// TIA Portal project "Forno" (V14)

(* hardware
DEVICE "S7-1200 station_1"  S7-1200 Station
   slot 0: "Rack_0"  Rack  V1.0
   slot 1: "PLC_1"  CPU 1214C DC/DC/DC  6ES7 214-1AG31-0XB0  V3.0
*)

// ===== PLC "PLC_1"  CPU 1214C DC/DC/DC =====

VAR_GLOBAL   // PLC tag table "Default tag table"
   "Pressostato_alta" AT %M0.0 : Bool;
   "Pressostato_baixa" AT %M0.1 : Bool;
   "Fluxo_exaust" AT %M0.2 : Bool;
   "Fluxo_forc" AT %M0.3 : Bool;
   "porta_closed" AT %M0.4 : Bool;
   "porta_opened" AT %M0.5 : Bool;
   "chama_piloto" AT %M0.6 : Bool;
   "chama_pricipal" AT %M0.7 : Bool;
   "Relay_chama_ok" AT %M1.0 : Bool;
   "Vent_exaust" AT %Q0.0 : Bool;
   "Vent_forc" AT %Q0.1 : Bool;
   "open_porta" AT %Q0.2 : Bool;
   "close_porta" AT %Q0.3 : Bool;
   "Valv_controle" AT %Q0.4 : Bool;
   "Bloqueio" AT %Q0.5 : Bool;
   "Relay_chama_comando" AT %Q0.6 : Bool;
   "intertravamentos" AT %M1.1 : Bool;
   "botao_on" AT %M1.2 : Bool;
   "partida_ok" AT %M1.3 : Bool;
   "purga_ok" AT %M1.4 : Bool;
   "ignicao" AT %M1.6 : Bool;
   "tentativa1" AT %M1.7 : Bool;
   "tentativa2" AT %M2.0 : Bool;
   "tentativa3" AT %M2.1 : Bool;
END_VAR

// folder: System blocks/Program resources

DATA_BLOCK "IEC_Timer_0_DB"   // DB1
{ S7_Optimized_Access := 'TRUE' }
AUTHOR : Simatic
FAMILY : IEC
NAME : IEC_TMR
VERSION : 1.0
// stored: InstanceOfName IEC_TIMER
"IEC_TIMER"
BEGIN
END_DATA_BLOCK

DATA_BLOCK "IEC_Timer_0_DB_1"   // DB2
{ S7_Optimized_Access := 'TRUE' }
AUTHOR : Simatic
FAMILY : IEC
NAME : IEC_TMR
VERSION : 1.0
// stored: InstanceOfName IEC_TIMER
"IEC_TIMER"
BEGIN
END_DATA_BLOCK

DATA_BLOCK "IEC_Timer_0_DB_3"   // DB4
{ S7_Optimized_Access := 'TRUE' }
AUTHOR : Simatic
FAMILY : IEC
NAME : IEC_TMR
VERSION : 1.0
// stored: InstanceOfName IEC_TIMER
"IEC_TIMER"
BEGIN
END_DATA_BLOCK

DATA_BLOCK "IEC_Timer_0_DB_4"   // DB5
{ S7_Optimized_Access := 'TRUE' }
AUTHOR : Simatic
FAMILY : IEC
NAME : IEC_TMR
VERSION : 1.0
// stored: InstanceOfName IEC_TIMER
"IEC_TIMER"
BEGIN
END_DATA_BLOCK

// folder: (top level)

FUNCTION "Purga" : Void   // FC1, LAD
{ S7_Optimized_Access := 'TRUE' }
VERSION : 0.1
BEGIN

REGION Network 1
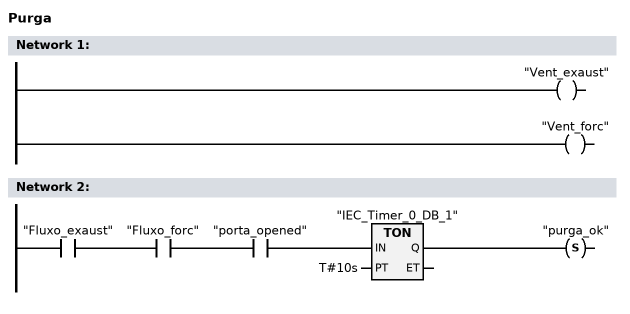
   RUNG wire#powerrail
      Coil( "Vent_exaust" )
   END_RUNG
   RUNG wire#powerrail
      Coil( "Vent_forc" )
   END_RUNG
   // the same network as SCL:
   "Vent_exaust" := TRUE;
   "Vent_forc" := TRUE;
END_REGION

REGION Network 2
   "IEC_Timer_0_DB_1".TON(IN := "Fluxo_exaust" AND "Fluxo_forc" AND "porta_opened", PT := T#10s);
   IF "IEC_Timer_0_DB_1".Q THEN "purga_ok" := TRUE; END_IF;
END_REGION
END_FUNCTION

ORGANIZATION_BLOCK "Main"   // OB1, LAD, ProgramCycle
TITLE = "Main Program Sweep (Cycle)"
{ S7_Optimized_Access := 'TRUE' }
VERSION : 0.1
BEGIN

REGION Network 1
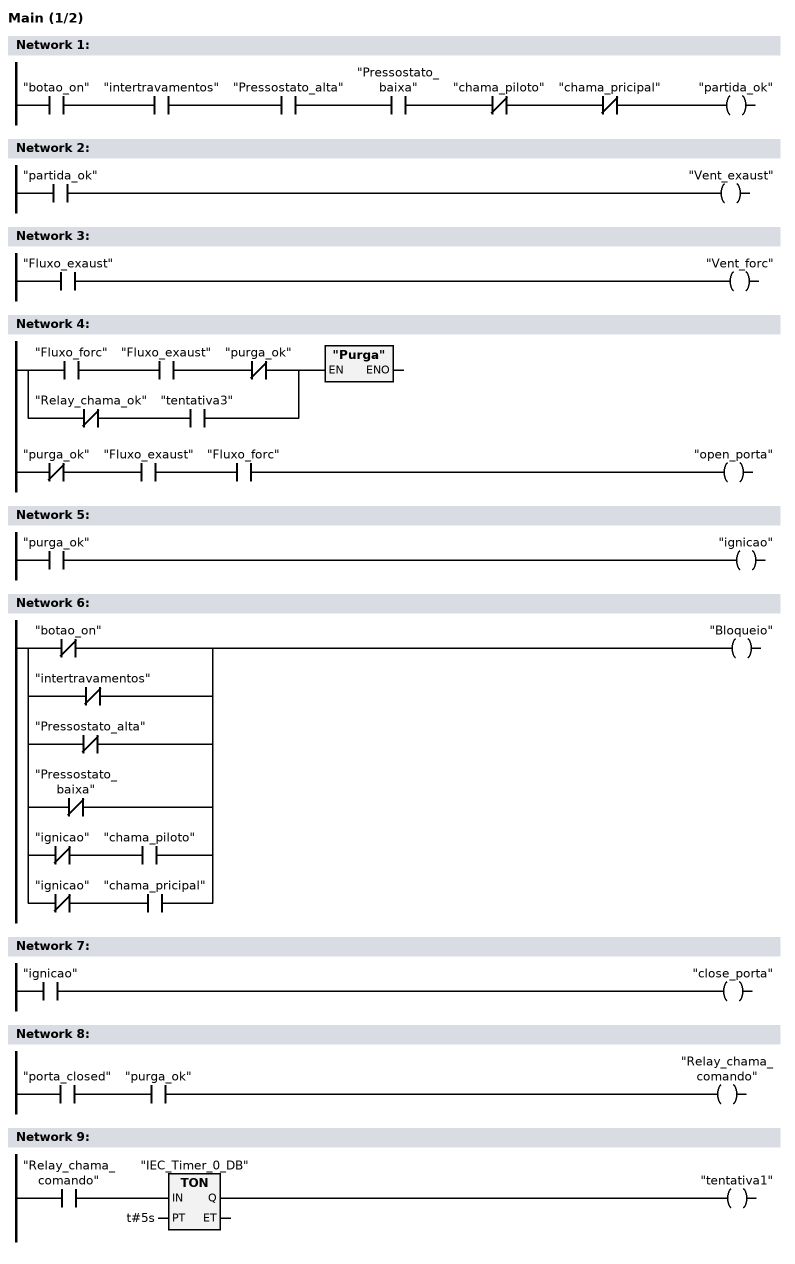
   RUNG wire#powerrail
      Contact( "botao_on" )
      Contact( "intertravamentos" )
      Contact( "Pressostato_alta" )
      Contact( "Pressostato_baixa" )
      I_Contact( "chama_piloto" )
      I_Contact( "chama_pricipal" )
      Coil( "partida_ok" )
   END_RUNG
   // the same network as SCL:
   "partida_ok" := "botao_on" AND "intertravamentos" AND "Pressostato_alta" AND "Pressostato_baixa" AND NOT "chama_piloto" AND NOT "chama_pricipal";
END_REGION

REGION Network 2
   RUNG wire#powerrail
      Contact( "partida_ok" )
      Coil( "Vent_exaust" )
   END_RUNG
   // the same network as SCL:
   "Vent_exaust" := "partida_ok";
END_REGION

REGION Network 3
   RUNG wire#powerrail
      Contact( "Fluxo_exaust" )
      Coil( "Vent_forc" )
   END_RUNG
   // the same network as SCL:
   "Vent_forc" := "Fluxo_exaust";
END_REGION

REGION Network 4
   RUNG wire#powerrail
      Contact( "Fluxo_forc" )
      Contact( "Fluxo_exaust" )
      I_Contact( "purga_ok" )
      wire#w1
      "Purga"()
   END_RUNG
   RUNG wire#powerrail
      I_Contact( "Relay_chama_ok" )
      Contact( "tentativa3" )
   END_RUNG wire#w1
   RUNG wire#powerrail
      I_Contact( "purga_ok" )
      Contact( "Fluxo_exaust" )
      Contact( "Fluxo_forc" )
      Coil( "open_porta" )
   END_RUNG
   // the same network as SCL:
   IF ("Fluxo_forc" AND "Fluxo_exaust" AND NOT "purga_ok") OR (NOT "Relay_chama_ok" AND "tentativa3") THEN
       "Purga"();
   END_IF;
   "open_porta" := NOT "purga_ok" AND "Fluxo_exaust" AND "Fluxo_forc";
END_REGION

REGION Network 5
   RUNG wire#powerrail
      Contact( "purga_ok" )
      Coil( "ignicao" )
   END_RUNG
   // the same network as SCL:
   "ignicao" := "purga_ok";
END_REGION

REGION Network 6
   RUNG wire#powerrail
      I_Contact( "botao_on" )
      wire#w1
      Coil( "Bloqueio" )
   END_RUNG
   RUNG wire#powerrail
      I_Contact( "intertravamentos" )
   END_RUNG wire#w1
   RUNG wire#powerrail
      I_Contact( "Pressostato_alta" )
   END_RUNG wire#w1
   RUNG wire#powerrail
      I_Contact( "Pressostato_baixa" )
   END_RUNG wire#w1
   RUNG wire#powerrail
      I_Contact( "ignicao" )
      Contact( "chama_piloto" )
   END_RUNG wire#w1
   RUNG wire#powerrail
      I_Contact( "ignicao" )
      Contact( "chama_pricipal" )
   END_RUNG wire#w1
   // the same network as SCL:
   "Bloqueio" := NOT "botao_on" OR NOT "intertravamentos" OR NOT "Pressostato_alta" OR NOT "Pressostato_baixa" OR (NOT "ignicao" AND "chama_piloto") OR (NOT "ignicao" AND "chama_pricipal");
END_REGION

REGION Network 7
   RUNG wire#powerrail
      Contact( "ignicao" )
      Coil( "close_porta" )
   END_RUNG
   // the same network as SCL:
   "close_porta" := "ignicao";
END_REGION

REGION Network 8
   RUNG wire#powerrail
      Contact( "porta_closed" )
      Contact( "purga_ok" )
      Coil( "Relay_chama_comando" )
   END_RUNG
   // the same network as SCL:
   "Relay_chama_comando" := "porta_closed" AND "purga_ok";
END_REGION

REGION Network 9
   "IEC_Timer_0_DB".TON(IN := "Relay_chama_comando", PT := t#5s);
   "tentativa1" := "IEC_Timer_0_DB".Q;
END_REGION

REGION Network 10
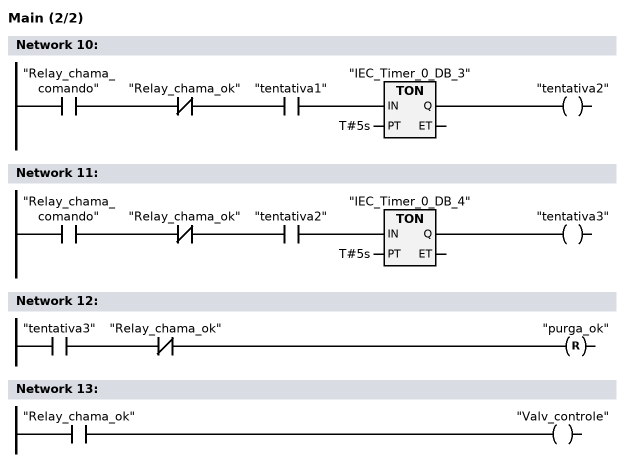
   "IEC_Timer_0_DB_3".TON(IN := "Relay_chama_comando" AND NOT "Relay_chama_ok" AND "tentativa1", PT := T#5s);
   "tentativa2" := "IEC_Timer_0_DB_3".Q;
END_REGION

REGION Network 11
   "IEC_Timer_0_DB_4".TON(IN := "Relay_chama_comando" AND NOT "Relay_chama_ok" AND "tentativa2", PT := T#5s);
   "tentativa3" := "IEC_Timer_0_DB_4".Q;
END_REGION

REGION Network 12
   RUNG wire#powerrail
      Contact( "tentativa3" )
      I_Contact( "Relay_chama_ok" )
      R_Coil( "purga_ok" )
   END_RUNG
   // the same network as SCL:
   IF "tentativa3" AND NOT "Relay_chama_ok" THEN "purga_ok" := FALSE; END_IF;
END_REGION

REGION Network 13
   RUNG wire#powerrail
      Contact( "Relay_chama_ok" )
      Coil( "Valv_controle" )
   END_RUNG
   // the same network as SCL:
   "Valv_controle" := "Relay_chama_ok";
END_REGION
END_ORGANIZATION_BLOCK

ORGANIZATION_BLOCK "Startup"   // OB100, LAD, Startup
TITLE = "Complete Restart"
{ S7_Optimized_Access := 'TRUE' }
VERSION : 0.1
   VAR_INPUT
      LostRetentive : Bool;   // True if retentive data are lost
      LostRTC : Bool;   // True if date and time are lost
   END_VAR
BEGIN

REGION Network 1
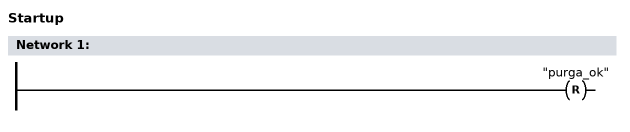
   RUNG wire#powerrail
      R_Coil( "purga_ok" )
   END_RUNG
   // the same network as SCL:
   "purga_ok" := FALSE;
END_REGION
END_ORGANIZATION_BLOCK